PROGRAM EMS_Start
VAR
	RESET: BOOL;
END_VAR

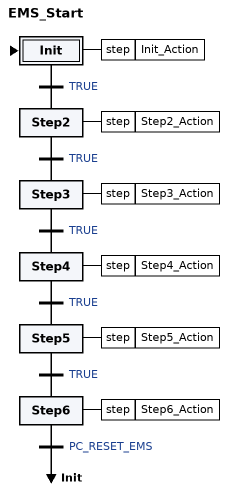
INITIAL_STEP Init:
    Init_Action(N);  // step action
END_STEP
TRANSITION FROM Init TO Step2
    := TRUE;
END_TRANSITION
STEP Step2:
    Step2_Action(N);  // step action
END_STEP
TRANSITION FROM Step2 TO Step3
    := TRUE;
END_TRANSITION
STEP Step3:  // min time t#1s
    Step3_Action(N);  // step action
END_STEP
TRANSITION FROM Step3 TO Step4
    := TRUE;
END_TRANSITION
STEP Step4:
    Step4_Action(N);  // step action
END_STEP
TRANSITION FROM Step4 TO Step5
    := TRUE;
END_TRANSITION
STEP Step5:  // min time t#1s
    Step5_Action(N);  // step action
END_STEP
TRANSITION FROM Step5 TO Step6
    := TRUE;
END_TRANSITION
STEP Step6:
    Step6_Action(N);  // step action
END_STEP
TRANSITION FROM Step6 TO Init
    := PC_RESET_EMS;
END_TRANSITION

ACTION Step5_Action:
EMS_RESET:=TRUE;
END_ACTION

ACTION Step4_Action:
EMS_ACK:=FALSE;
END_ACTION

ACTION Step6_Action:
EMS_RESET:=FALSE;
END_ACTION

ACTION Init_Action:

	EMS_RUN:=FALSE;
	EMS_ACK:=FALSE;
	EMS_RESET:=FALSE;

	RESET:=FALSE;
END_ACTION

ACTION Step2_Action:
EMS_RUN:=TRUE;
END_ACTION

ACTION Step3_Action:
EMS_ACK:=TRUE;
END_ACTION

END_PROGRAM

(* stored: Version 1.1.0.1, ProductVersion 3.1.0.26
   POU EMS_Start: Id {c3e91596-8672-4902-b857-6f89842e7b5b}
   Action Step5_Action: Id {20913055-fb41-44b8-bdfc-b70a259fe406}
   Action Step4_Action: Id {5ab81576-f187-4d5a-8a61-cd3ec997fb76}
   Action Step6_Action: Id {8a079c24-cc92-4ee8-a579-12ffe99100b5}
   Action Init_Action: Id {8e92a162-e3b9-4948-abc6-c3f57190bd23}
   Action Step2_Action: Id {ab97de92-f771-4732-9165-a27aaeac48d0}
   Action Step3_Action: Id {b1faf266-8366-4b8c-b0c2-07a3b905f0de} *)
